{attribute 'qualified_only'}
{attribute 'strict'}
{attribute 'to_string'}
TYPE E_OperatorInstruction :
(
    None := 0,
    LoadInitialPuck := 10,
    WaitPuckLocking := 20,
    RemovePassedPart := 30,
    RemoveFailedPart := 40,
    PlacePartInRejectBin := 50,
    RemoveReleasedPuck := 60,
    LoadNewPuck := 70,
    LoadPart := 80,
    ReadyToIndex := 90,
    ReadyToIndexEmpty := 100,
    TableIndexing := 110,
    RestoreUnexpectedlyRemovedPuck := 120
);
END_TYPE

(* stored: Version 1.1.0.1, ProductVersion 3.1.4026.18
   DUT E_OperatorInstruction: Id {57eaeef2-bb4f-4263-b7b1-def9c520612d} *)
